// TIA Portal V16 export
// export: Created 2024-06-24T15:42:28.0355103Z, ExportSetting WithDefaults, DisplayName Totally Integrated Automation Portal, DisplayVersion V16, DisplayName TIA Portal Version Control Interface, DisplayVersion V16, DisplayName TIA Portal Openness, DisplayVersion V16, DisplayName STEP 7 Professional, DisplayVersion V16, DisplayName STEP 7 Safety, DisplayVersion V16, DisplayName WinCC Advanced, DisplayVersion V16
ORGANIZATION_BLOCK "OB_PickAndPlace"   // OB127, LAD, ProgramCycle
TITLE = "Main Program Sweep (Cycle)"
{ S7_Optimized_Access := 'TRUE' }
VERSION : 0.1
// stored: AutoNumber true, IsIECCheckEnabled false, SetENOAutomatically false
   VAR_INPUT
      Initial_Call : Bool;   // Initial call of this OB
      Remanence : Bool;   // =True, if remanent data are available
   END_VAR
   VAR_TEMP   // added for the SCL form of the ladder/FBD networks
      _w1 : Bool;
   END_VAR
BEGIN

REGION Network 1
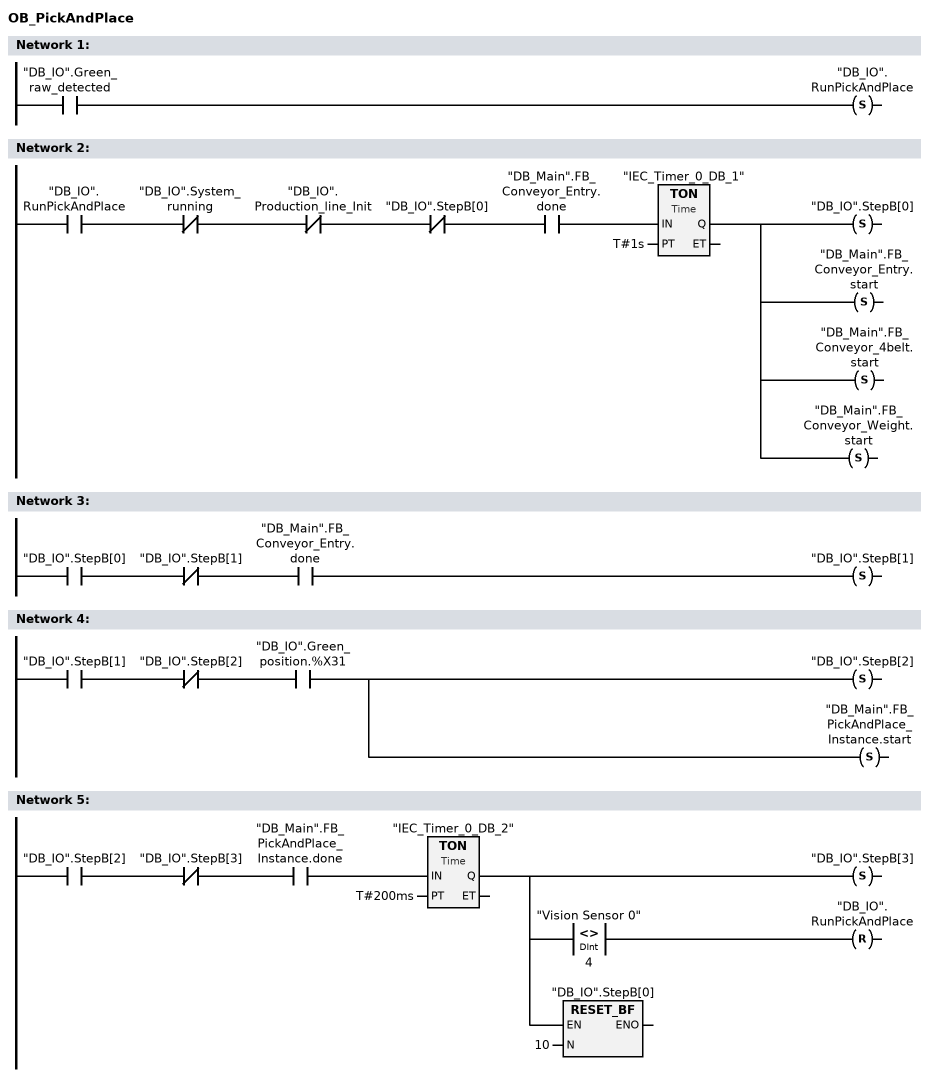
   RUNG wire#powerrail
      Contact( "DB_IO".Green_raw_detected )
      S_Coil( "DB_IO".RunPickAndPlace )
   END_RUNG
   // the same network as SCL:
   IF "DB_IO".Green_raw_detected THEN "DB_IO".RunPickAndPlace := TRUE; END_IF;
END_REGION

REGION Network 2
   RUNG wire#powerrail
      Contact( "DB_IO".RunPickAndPlace )
      I_Contact( "DB_IO".System_running )
      I_Contact( "DB_IO".Production_line_Init )
      I_Contact( "DB_IO".StepB[0] )
      Contact( "DB_Main".FB_Conveyor_Entry.done )
      { S7_Templates := "time_type := Time" } "IEC_Timer_0_DB_1".TON(pt := T#1s, et =>)
      wire#w1
      S_Coil( "DB_IO".StepB[0] )
   END_RUNG
   RUNG wire#w1
      S_Coil( "DB_Main".FB_Conveyor_Entry.start )
   END_RUNG
   RUNG wire#w1
      S_Coil( "DB_Main".FB_Conveyor_4belt.start )
   END_RUNG
   RUNG wire#w1
      S_Coil( "DB_Main".FB_Conveyor_Weight.start )
   END_RUNG
   // the same network as SCL:
   "IEC_Timer_0_DB_1".TON(IN := "DB_IO".RunPickAndPlace AND NOT "DB_IO".System_running AND NOT "DB_IO".Production_line_Init AND NOT "DB_IO".StepB[0] AND "DB_Main".FB_Conveyor_Entry.done,
                          PT := T#1s);
   IF "IEC_Timer_0_DB_1".Q THEN
       "DB_IO".StepB[0] := TRUE;
       "DB_Main".FB_Conveyor_Entry.start := TRUE;
       "DB_Main".FB_Conveyor_4belt.start := TRUE;
       "DB_Main".FB_Conveyor_Weight.start := TRUE;
   END_IF;
END_REGION

REGION Network 3
   RUNG wire#powerrail
      Contact( "DB_IO".StepB[0] )
      I_Contact( "DB_IO".StepB[1] )
      Contact( "DB_Main".FB_Conveyor_Entry.done )
      S_Coil( "DB_IO".StepB[1] )
   END_RUNG
   // the same network as SCL:
   IF "DB_IO".StepB[0] AND NOT "DB_IO".StepB[1] AND "DB_Main".FB_Conveyor_Entry.done THEN
       "DB_IO".StepB[1] := TRUE;
   END_IF;
END_REGION

REGION Network 4
   RUNG wire#powerrail
      Contact( "DB_IO".StepB[1] )
      I_Contact( "DB_IO".StepB[2] )
      Contact( "DB_IO".Green_position.%X31 )
      wire#w1
      S_Coil( "DB_IO".StepB[2] )
   END_RUNG
   RUNG wire#w1
      S_Coil( "DB_Main".FB_PickAndPlace_Instance.start )
   END_RUNG
   // the same network as SCL:
   #_w1 := "DB_IO".StepB[1] AND NOT "DB_IO".StepB[2] AND "DB_IO".Green_position.%X31;
   IF #_w1 THEN
       "DB_IO".StepB[2] := TRUE;
       "DB_Main".FB_PickAndPlace_Instance.start := TRUE;
   END_IF;
END_REGION

REGION Network 5
   // no SCL statement known for RBitfield: written as a call
   "IEC_Timer_0_DB_2".TON(IN := "DB_IO".StepB[2] AND NOT "DB_IO".StepB[3] AND "DB_Main".FB_PickAndPlace_Instance.done,
                          PT := T#200ms);
   IF "IEC_Timer_0_DB_2".Q THEN "DB_IO".StepB[3] := TRUE; END_IF;
   IF "IEC_Timer_0_DB_2".Q AND ("Vision Sensor 0" <> 4) THEN "DB_IO".RunPickAndPlace := FALSE; END_IF;
   IF "IEC_Timer_0_DB_2".Q THEN RESET_BF(operand := "DB_IO".StepB[0], n := 10); END_IF;
END_REGION
END_ORGANIZATION_BLOCK
